Fanuc KAREL source: kf00100.KL

-- PROVISIONAL review KL for V770-1; original PC SHA256 a0dcccf48a69b4e875bea283d574a23e16dae1b3826c0b498bc03a8a04a542a8
-- Incomplete behavior may be omitted. Consult companion uncertainty JSON. Do not deploy.
PROGRAM KF00100
%NOLOCKGROUP
BEGIN
  -- UNRESOLVED_PC offsets 5-16; opcodes 2E,23
  -- UNRESOLVED_PC offsets 21-32; opcodes 2E,23
  -- UNRESOLVED_PC offsets 37-63; opcodes 27,27,9D,22,1C,22,27,9D,31
  -- UNRESOLVED_PC offsets 68-72; opcodes 7F
END KF00100
